{attribute 'qualified_only'}
{attribute 'strict'}
TYPE E_LogStatusReport_Type :
(
	General:=	0,
	Speed,
	Eng,
	EFS

);
END_TYPE

(* stored: Version 1.1.0.1, ProductVersion 3.1.4024.3
   DUT E_LogStatusReport_Type: Id {49bd01b7-3c22-0170-3c16-33642ff8348b} *)
